TYPE E_ConveyorState :
   (
       Stopped := 0,
       Starting := 1,
       Running := 2,
       Faulted := 3
   ) DINT;
   END_TYPE

(* stored: Version 1.1.0.1, ProductVersion 3.1.4026.18
   DUT E_ConveyorState: Id {1faa1491-96b3-4817-bd7d-d45e0541cd35} *)
